// TIA Portal V18 export
DATA_BLOCK "material Data Recipe"   // DB331
{ S7_Optimized_Access := 'TRUE' }
VERSION : 0.1
// stored: AutoNumber true, DBAccessibleFromOPCUA true, IsOnlyStoredInLoadMemory false, IsRetainMemResEnabled false, IsWriteProtectedInAS false, MemoryReserve 100
   VAR
      "Material 1" : Struct
         "Mixing ratio" : Real := 25.0;
         "Name A" : String[20] := 'resin1';
         "Name B" : String[20] := 'hardener1';
         "Density A" : Real;
         "Density B" : Real;
         "Viscosity A" : Real;
         "Vsicosity B" : Real;
         "A+" : String[21];
         "Name A+B" : String[42];
      END_STRUCT;
   END_VAR
   VAR RETAIN
      Selection : Int;
   END_VAR
   VAR
      "Selected material" : String;
   END_VAR
   VAR RETAIN
      "+symbol" : String := '+';
   END_VAR
BEGIN
END_DATA_BLOCK
